TYPE "IPC_Msg_Log_PAR"
VERSION : 0.1
// Block: IPC_Msg_Log_PAR
   STRUCT
      Id : DInt;
      timestamp : String;
      topic : UDInt;
      payLoad_1 : String;
      payLoad_2 : String;
      payLoad_3 : String;
      payLoad_4 : String;
      payLoad_5 : String;
   END_STRUCT;

END_TYPE
